Universal Robots PolyScope program: EGH80_is_gripped_test.urp

Program EGH80_is_gripped_test (installation=default directory=/programs/Tests createdIn=5.9.1.1031110 lastSavedIn=5.9.1.1031110 robotSerialNumber=20185500256)
Calibrated DH parameters: a=[0.000163, -0.146131, -0.38577, 0.000126, -0.000021, 0]; d=[0.161954, 188.306531, -157.478086, -30.695088, 0.099716, 0.099628]; alpha=[1.569701, -0.00212, 0.002263, 1.570438, -1.570123, 0]; deltaTheta=[0, -1.219859, 7.681919, -0.178877, -0.000001, 0]
BeforeStart
  Call EGH80_connect
Robot Program (runOnlyOnce=true)
  URCap EGH Grip (EGH-SCHUNK, SCHUNK GmbH & Co. KG) dataModel(actionType=false)
  is_gripped := EGH80_grip()
SubProgram  [hidden by the author, left out]
SubProgram EGH80_grip [hidden by the author, left out]
SubProgram EGH80_connect [hidden by the author, left out]
